VAR_GLOBAL
	maxSimulationTorque: INT;
	maxSimulationVelocity: INT;
	Actual_Velocity: LREAL;
	ActualTorque AT %I*: LREAL;
	SetVelocity: INT;
	SetTorque: INT;
END_VAR

(* stored: Version 1.1.0.1, ProductVersion 3.1.4024.4
   GVL GVL: Id {dd000a01-6078-422b-9413-b0ea23df6a4b} *)
